FUNCTION_BLOCK Mc2StopTask EXTENDS Mc2MotionTask IMPLEMENTS I_Mc2MotionTask
VAR
	McHalt		  : Tc2_MC2.MC_Halt;
	_McBufferMode : Tc2_MC2.MC_BufferMode;
	_MoveOptions  : Tc2_MC2.ST_MoveOptions;
END_VAR

PROPERTY BufferMode : REFERENCE TO MC_BufferMode
GET
BufferMode REF= _McBufferMode;
END_GET
END_PROPERTY

{attribute 'monitoring' := 'call'}
PROPERTY Busy : BOOL
GET
Busy := McHalt.Busy;
END_GET
END_PROPERTY

METHOD CyclicLogic
McHalt(Axis			:= _Axis.Axis,
	   Deceleration := _Axis.Deceleration,
	   Jerk			:= _Axis.Jerk,
	   BufferMode	:= _McBufferMode,
	   Options		:= _MoveOptions);

McHalt.Execute := FALSE;
END_METHOD

{attribute 'monitoring' := 'call'}
PROPERTY Error : BOOL
GET
Error := McHalt.Error;
END_GET
END_PROPERTY

{attribute 'monitoring' := 'call'}
PROPERTY ErrorId : UDINT
GET
ErrorId := McHalt.ErrorID;
END_GET
END_PROPERTY

METHOD Execute : BOOL
McHalt(Axis			:= _Axis.Axis,
	   Execute		:= TRUE,
	   Deceleration := _Axis.Deceleration,
	   Jerk			:= _Axis.Jerk,
	   BufferMode	:= _McBufferMode,
	   Options		:= _MoveOptions);

Execute := TRUE;
END_METHOD

PROPERTY MoveOptions : REFERENCE TO ST_MoveOptions
GET
MoveOptions REF= _MoveOptions;
END_GET
END_PROPERTY

END_FUNCTION_BLOCK

(* stored: Version 1.1.0.1, ProductVersion 3.1.4026.20
   POU Mc2StopTask: Id {9a6b8d8e-a659-47bd-980a-87ba4fadf676}, SpecialFunc None
   Property BufferMode: Id {f011db3d-f3e3-4de2-bb74-8bb86a10aaa5}
   Get Get: Id {072b694e-6637-403d-9d5a-8e27438a46ae}
   Property Busy: Id {d81b57df-1d5a-4e22-a700-80e24d83bf48}
   Get Get: Id {43b8abd4-d74d-46a6-8b7c-f0b79805720a}
   Method CyclicLogic: Id {9e96c630-e29c-480d-a2a3-bd48eaa0b545}
   Property Error: Id {a036a230-83af-49dd-8d79-11a5509a5434}
   Get Get: Id {1c7e877f-b790-4bbb-9b4c-1774ee7e65a1}
   Property ErrorId: Id {687e7b07-e3b6-4ce9-bd4f-b06c77b74f11}
   Get Get: Id {756ae493-9f7f-4f18-a93d-f87fe03e9ed2}
   Method Execute: Id {cf9ec3ae-3953-44dd-96a8-6aac0346277b}
   Property MoveOptions: Id {1144f10b-404d-49b2-9659-a36e49a5fbe2}
   Get Get: Id {82078bdd-a39c-4f83-a658-84d97b4caad1} *)
